(* IEC 61131-3 sources: ladder-web-ide/backend/tests/fixtures/iec2c_saidas/entrada, 3 files *)

(* ---- erro_sintaxe.st ---- *)
PROGRAM prog0
  VAR
    a : BOOL
  END_VAR
  a := TRUE;
END_PROGRAM

CONFIGURATION Config0
  RESOURCE Res0 ON PLC
    TASK task0(INTERVAL := T#20ms, PRIORITY := 0);
    PROGRAM instance0 WITH task0 : prog0;
  END_RESOURCE
END_CONFIGURATION

(* ---- tipo_incompativel.st ---- *)
PROGRAM prog0
  VAR
    a : BOOL;
    b : INT;
  END_VAR
  a := b;
END_PROGRAM

CONFIGURATION Config0
  RESOURCE Res0 ON PLC
    TASK task0(INTERVAL := T#20ms, PRIORITY := 0);
    PROGRAM instance0 WITH task0 : prog0;
  END_RESOURCE
END_CONFIGURATION

(* ---- variavel_nao_declarada.st ---- *)
PROGRAM prog0
  VAR
    a : BOOL;
  END_VAR
  b := TRUE;
END_PROGRAM

CONFIGURATION Config0
  RESOURCE Res0 ON PLC
    TASK task0(INTERVAL := T#20ms, PRIORITY := 0);
    PROGRAM instance0 WITH task0 : prog0;
  END_RESOURCE
END_CONFIGURATION
